Fanuc KAREL source: INSERT_NODE.kl

PROGRAM T
%NOLOCKGROUP
VAR
 v0 : PATH
 v1 : INTEGER
 v2 : INTEGER
BEGIN
 INSERT_NODE(v0, v1, v2)
END T
